FUNCTION_BLOCK GenericCylinderModelType1 (* Composite Function Block Type *)
  (* Standard: 61499-2 *)
  (* Version 0.0, 12/5/2011, XPMUser, nxtControl GmbH, template *)
  PACKAGE Main;
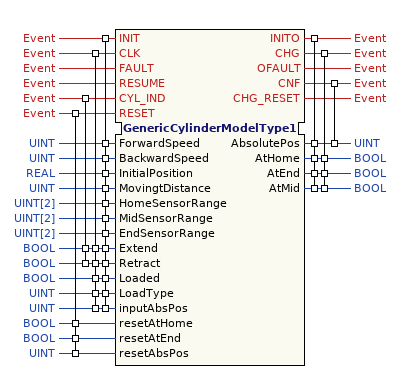
  EVENT_INPUT
    INIT WITH ForwardSpeed, BackwardSpeed, Extend, Retract, HomeSensorRange, EndSensorRange, InitialPosition, LoadType, MovingtDistance, Loaded, MidSensorRange, inputAbsPos; (* Initialization Request *)
    CLK WITH Extend, Retract, Loaded, LoadType, inputAbsPos; (* Clock signal *)
    FAULT;
    RESUME;
    CYL_IND WITH Extend, Retract;
    RESET WITH resetAtHome, resetAtEnd, resetAbsPos;
  END_EVENT
  EVENT_OUTPUT
    INITO WITH AbsolutePos, AtHome, AtEnd, AtMid; (* Initialization Confirm *)
    CHG WITH AtEnd, AtHome, AtMid; (* Indicate data outputs changed *)
    OFAULT;
    CNF WITH AbsolutePos;
    CHG_RESET;
  END_EVENT
  VAR_INPUT
    ForwardSpeed : UINT; (* Forward speed *)
    BackwardSpeed : UINT; (* Backward speed *)
    InitialPosition : REAL; (* Initial position *)
    MovingtDistance : UINT; (* Moving distance *)
    HomeSensorRange : ARRAY [0..1] OF UINT; (* Detection range of home sensor *)
    MidSensorRange : ARRAY [0..1] OF UINT; (* Detection range of home sensor *)
    EndSensorRange : ARRAY [0..1] OF UINT; (* Detection range of end sensor *)
    Extend : BOOL;
    Retract : BOOL;
    Loaded : BOOL;
    LoadType : UINT;
    inputAbsPos : UINT;
    resetAtHome : BOOL;
    resetAtEnd : BOOL;
    resetAbsPos : UINT;
  END_VAR
  VAR_OUTPUT
    AbsolutePos : UINT; (* Current position *)
    AtHome : BOOL; (* Detected at home position *)
    AtEnd : BOOL; (* Detected at end position *)
    AtMid : BOOL;
  END_VAR
  FBS
    MoveStatus : MovingStatus;
    Home : RangeSensor;
    Middle : RangeSensor;
    End : RangeSensor;
    Position : LinearMotionLoad;
  END_FBS
  EVENT_CONNECTIONS
    INIT TO MoveStatus.INIT;
    FAULT TO MoveStatus.FAULT;
    RESUME TO MoveStatus.RESUME;
    MoveStatus.INITO TO Position.INIT;
    Position.INITO TO Home.INIT;
    Home.INITO TO Middle.INIT;
    Middle.INITO TO End.INIT;
    End.INITO TO INITO;
    Position.CHG TO CNF;
    MoveStatus.OFAULT TO OFAULT;
    Position.CHG TO Home.CLK;
    RESET TO Position.RESET;
    Middle.CHG TO End.CLK;
    Home.CHG TO Middle.CLK;
    End.CHG TO CHG;
    End.CHG_RESET TO CHG_RESET;
    Middle.CHG_RESET TO End.RESET;
    Home.CHG_RESET TO Middle.RESET;
    Position.CHG_RESET TO Home.RESET;
    CLK TO MoveStatus.CLK;
    MoveStatus.CHG TO Position.CLK;
    MoveStatus.OFAULT TO Position.CLK;
  END_CONNECTIONS
  DATA_CONNECTIONS
    MoveStatus.C_FWD TO Position.MoveForwards;
    MoveStatus.C_BWD TO Position.MoveBackwards;
    Loaded TO Position.Loaded;
    LoadType TO Position.LoadType;
    Retract TO MoveStatus.Retract;
    Extend TO MoveStatus.Extend;
    EndSensorRange TO End.Zone;
    HomeSensorRange TO Home.Zone;
    Position.RelativePos TO Middle.Position;
    Position.RelativePos TO End.Position;
    Home.Detected TO AtHome;
    Middle.Detected TO AtMid;
    End.Detected TO AtEnd;
    ForwardSpeed TO Position.ForwardSpeed;
    BackwardSpeed TO Position.BackwardSpeed;
    InitialPosition TO Position.InitialPosition;
    MovingtDistance TO Position.MovingDistance;
    Position.AbsolutePos TO AbsolutePos;
    Position.RelativePos TO Home.Position;
    MidSensorRange TO Middle.Zone;
    inputAbsPos TO Position.inputAbsPos;
    resetAtHome TO Position.resetAtHome;
    resetAtEnd TO Position.resetAtEnd;
    resetAbsPos TO Position.resetAbsPos;
  END_CONNECTIONS
END_FUNCTION_BLOCK
